INTERFACE IOutput EXTENDS __SYSTEM.IQueryInterface

END_INTERFACE

(* stored: Version 1.1.0.1, ProductVersion 3.1.4024.12
   Itf IOutput: Id {66cf7dfe-1a8a-4840-bc34-49638d73d6ae} *)
